// TIA Portal V19 export
TYPE "lexchangetray_typeUnEmn_toRollerFeedback"
// Type: Bool
// stored: Access Published
   STRUCT
      inFeedEnabled : Bool;   // Manual mode parameters for axis control interface
      outFeeding : Bool;   // Manual mode parameters for axis control interface
   END_STRUCT;
END_TYPE
